FUNCTION_BLOCK Central_Server (* Basic Function Block Type *)
  (* Standard: 61499-2 *)
  (* Version 0.2, 2003-12-04, JHC, Rockwell Automation, Renamed for better indexing. *)
  (* Version 0.1, 2002-11-05, JHC, Rockwell Automation, Corrected missing ST element in Algorithm REQ. *)
  (* Version 0.0, 2000-05-30, JHC, Rockwell Automation *)
  (* Compiler header: package fb.rt.cs725; *)
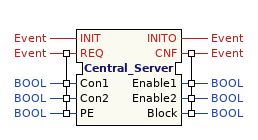
  EVENT_INPUT
    INIT; (* Initialization Request *)
    REQ WITH Con1, Con2, PE; (* Normal Execution Request *)
  END_EVENT
  EVENT_OUTPUT
    INITO; (* Initialization Confirm *)
    CNF WITH Enable2, Enable1, Block; (* Execution Confirmation *)
  END_EVENT
  VAR_INPUT
    Con1 : BOOL;
    Con2 : BOOL;
    PE : BOOL;
  END_VAR
  VAR_OUTPUT
    Enable1 : BOOL;
    Enable2 : BOOL;
    Block : BOOL;
  END_VAR
  VAR
    queue : ARRAY [0..2] OF INT;
    token : BOOL;
    test : ARRAY [0..2] OF INT;
  END_VAR
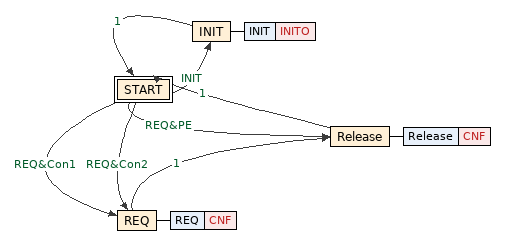
  EC_STATES
    START; (* Initial State *)
    INIT : INIT -> INITO; (* Initialization *)
    REQ : REQ -> CNF; (* Normal execution *)
    Release : Release -> CNF;
  END_STATES
  EC_TRANSITIONS
    START TO INIT := INIT;
    INIT TO START := 1;
    START TO REQ := REQ&Con1;
    START TO Release := REQ&PE;
    Release TO START := 1;
    REQ TO Release := 1;
    START TO REQ := REQ&Con2;
  END_TRANSITIONS
  ALGORITHM INIT IN Java: (* Initialization algorithm *)
Enable1.value=false;
Enable2.value=false;
  END_ALGORITHM
  ALGORITHM REQ IN Java: (* Normally executed algorithm *)
if (Con1.value){
if (queue.value[0] == null){
queue.value[0]='1';
}else if (queue.value[1] == null){
queue.value[1]=1;
}else{
queue.value[2]=1;
}
Enable1.value=true;
}
if (Con2.value){
if (queue.value[0] ==null){
queue.value[0]=2;
}else if (queue.value[1] ==null){
queue.value[1]=2;
}else{
queue.value[2]=2;
}
Enable2.value=true;
}
Block.value=true;
  END_ALGORITHM
  ALGORITHM Release IN Java:
if(PE.value){
token.value=true;
}
if(token.value){
if(queue.value[0]!=null){
if(queue.value[0]==1){
Enable1.value=true;
}else{
Enable2.value=true;
}
Block.value=false;
token.value=false;
queue.value[0]=queue.value[1];
queue.value[1]=queue.value[2];
queue.value[2]=null;
}
}
  END_ALGORITHM
END_FUNCTION_BLOCK
